{attribute 'strict'}
{attribute 'to_string'}
TYPE E_Robot_Programs :
(
	NoCommand			:= 0,
	Home				:= 1,
	Park				:= 2,
	Service				:= 3,
	VisePickUp_1_7 		:= 11,
	VisePutDown_1_7 	:= 12,
	VisePickUp_8_14		:= 13,
	VisePutDown_8_14	:= 14,
	VisePutDownToCnc_4 	:= 15,
	VisePickUpFromCnc_4	:= 16,
	VisePutDownToCnc_5	:= 17,
	VisePickUpFromCnc_5	:= 18
);
END_TYPE

(* stored: Version 1.1.0.1, ProductVersion 3.1.4024.11
   EnumerationTextList E_Robot_Programs: Id {5a2ec05a-b70c-4986-be60-01cf6850b16e} *)
